TYPE ST_DynSectorStatus :
STRUCT
	XtsRefData								: REFERENCE TO Tc3_XTS_Utility.ST_PositionInfo;
	HasInterference						: BOOL;
	TrackSectorBndryHead			: LREAL;
	TrackSectorBndryTail			: LREAL;
	TrackSectorCenterHead			: LREAL;
	TrackSectorCenterTail			: LREAL;	
	PartSectorBndryHead				: LREAL;
	PartSectorBndryTail				: LREAL;
	PartSectorCenterHead			: LREAL;
	PartSectorCenterTail			: LREAL;	
END_STRUCT
END_TYPE

(* stored: Version 1.1.0.1
   DUT ST_DynSectorStatus: Id {a98e7ea4-f570-0414-0e88-a9faaf2729e3} *)
